PROGRAM MAIN
VAR
END_VAR

END_PROGRAM

(* stored: Version 1.1.0.1
   POU MAIN: Id {61ca4f67-3f79-4581-90d6-7436e7374222} *)
